Staubli VAL3: unique.pgx

program unique(string& x_sResult[])
  local num l_nElement
  local bool l_bFound
  local num l_nBuffer
begin

  for l_nElement = 0 to size(lSplit.sString)-1
    l_bFound = false
    if l_nElement == 0
      append(x_sResult)
      x_sResult[size(x_sResult)-1] = lSplit.sString[l_nElement]
    else

      for l_nBuffer = 0 to size(x_sResult)-1
        if lSplit.sString[l_nElement] != x_sResult[l_nBuffer]
          l_bFound = false
        else
          // break out of for-loop
          l_bFound = true
          l_nBuffer = size(x_sResult)+1
        endIf

      endFor

      if l_bFound == false
        append(x_sResult)
        x_sResult[size(x_sResult)-1] = lSplit.sString[l_nElement]
      endIf

   endIf

  endFor

  delete(x_sResult[0])

end
